(* IEC 61131-3 sources: 2026_Projet_YGO_ExcavatriceDragage/TOOLS/TEST_AUTO_CI/RESULTS/TREUILS/tests, 2 files *)

(* ---- test_fb_bucket.st ---- *)
SETUP
VAR
    FB : FB_Bucket;
    BucketState : ST_BucketState;
END_VAR
END_SETUP

TEST 'Bucket : Enable=FALSE neutralise le pilotage benne'
    FB(Enable := FALSE, PowerContactorEngaged := TRUE, BucketState := BucketState);
    ASSERT_FALSE(FB.Ready, 'Ready doit etre FALSE sans Enable');
    ASSERT_FALSE(FB.M2_StartStop, 'M2_StartStop coupe');
END_TEST

(* ---- test_fb_winch.st ---- *)
SETUP
VAR
    FB_Safety : FB_Safety_Winch;
    FB_W : FB_Winch;
END_VAR
END_SETUP

TEST 'Safety_Winch : Enable=FALSE neutralise les autorisations'
    FB_Safety(Enable := FALSE, PowerContactorEngaged := TRUE);
    ASSERT_FALSE(FB_Safety.Ready, 'Ready doit etre FALSE sans Enable');
END_TEST

TEST 'Winch : Enable=FALSE neutralise les sorties'
    FB_W(Enable := FALSE, PowerContactorEngaged := TRUE);
    ASSERT_FALSE(FB_W.Ready, 'Ready doit etre FALSE sans Enable');
    ASSERT_FALSE(FB_W.RelayFwd, 'RelayFwd coupe');
    ASSERT_FALSE(FB_W.RelayRev, 'RelayRev coupe');
END_TEST
